FUNCTION_BLOCK Motion_Observer IMPLEMENTS ITF_Observer
VAR
	SystemSafetyState : INT;
END_VAR

METHOD Update : BOOL
VAR_INPUT
	TwinSAFEState : INT;
END_VAR
SystemSafetyState := TwinSAFEState;
END_METHOD

END_FUNCTION_BLOCK

(* stored: Version 1.1.0.1, ProductVersion 3.1.4024.12
   POU Motion_Observer: Id {740b309b-9ac9-459a-be4a-b6b2c942ba0a}, SpecialFunc None
   Method Update: Id {d0c5958a-729a-41c7-8e02-87338ae907e6} *)
